{attribute 'GeneratedUsingTerminal: EL3773-0000-0016'}
{attribute addProperty BoxType "EL3773-0000-0016"}
{attribute addProperty Id "I2_STATUSAT %I*I2_STATUS_B07533568"}
{attribute addProperty CRC "4153007013"}
{attribute addProperty Size "8"}
TYPE L2_Current_Status_F789DBA5 EXTENDS InputBase_8311D824 :
STRUCT
	{attribute addProperty Name "I2_STATUS"}
	I2_STATUS AT %I* : I2_STATUS_B0753356;
END_STRUCT
END_TYPE

(* stored: Version 1.2.0.0, ProductVersion 3.1.4024.9
   DUT L2_Current_Status_F789DBA5: Id {cc48dbca-bbb5-4687-ab72-bd92fabeb9a6} *)
